# EPICS substitutions: apps/svtCtrlApp/Db/crate_r1.substitutions
# SVT HFCB HV & LV wiener modules substitution file
#  for iseg (HV) MX is slot # 1-10
file iocsoftsvtAppsV/db/iseg.db {
pattern { HOST, MX }
  {"vmetlsvt1","7"}
  {"vmetlsvt1","8"}
}
#  for mpv (LV) MX is slot # 0-9
file iocsoftsvtAppsV/db/mpv.db {
   pattern { HOST, MX }
  {"vmetlsvt1","0"}
  {"vmetlsvt1","1"}
  {"vmetlsvt1","2"}
  {"vmetlsvt1","3"}
  {"vmetlsvt1","4"}
}
